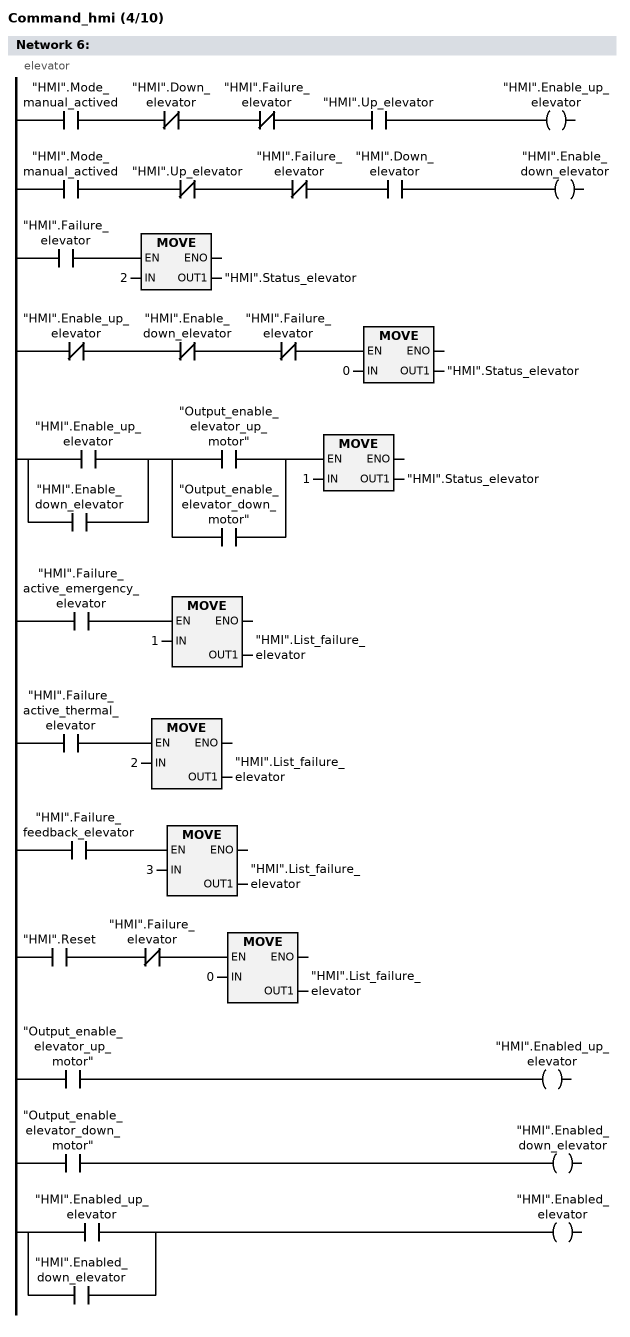
   RUNG wire#powerrail
      Contact( "HMI".Mode_manual_actived )
      I_Contact( "HMI".Down_elevator )
      I_Contact( "HMI".Failure_elevator )
      Contact( "HMI".Up_elevator )
      Coil( "HMI".Enable_up_elevator )
   END_RUNG
   RUNG wire#powerrail
      Contact( "HMI".Mode_manual_actived )
      I_Contact( "HMI".Up_elevator )
      I_Contact( "HMI".Failure_elevator )
      Contact( "HMI".Down_elevator )
      Coil( "HMI".Enable_down_elevator )
   END_RUNG
   RUNG wire#powerrail
      Contact( "HMI".Failure_elevator )
      Move(in := 2, out1 => "HMI".Status_elevator)
   END_RUNG
   RUNG wire#powerrail
      I_Contact( "HMI".Enable_up_elevator )
      I_Contact( "HMI".Enable_down_elevator )
      I_Contact( "HMI".Failure_elevator )
      Move(in := 0, out1 => "HMI".Status_elevator)
   END_RUNG
   RUNG wire#powerrail
      Contact( "HMI".Enable_up_elevator )
      wire#w1
      Contact( "Output_enable_elevator_up_motor" )
      wire#w2
      Move(in := 1, out1 => "HMI".Status_elevator)
   END_RUNG
   RUNG wire#powerrail
      Contact( "HMI".Enable_down_elevator )
   END_RUNG wire#w1
   RUNG wire#w1
      Contact( "Output_enable_elevator_down_motor" )
   END_RUNG wire#w2
   RUNG wire#powerrail
      Contact( "HMI".Failure_active_emergency_elevator )
      Move(in := 1, out1 => "HMI".List_failure_elevator)
   END_RUNG
   RUNG wire#powerrail
      Contact( "HMI".Failure_active_thermal_elevator )
      Move(in := 2, out1 => "HMI".List_failure_elevator)
   END_RUNG
   RUNG wire#powerrail
      Contact( "HMI".Failure_feedback_elevator )
      Move(in := 3, out1 => "HMI".List_failure_elevator)
   END_RUNG
   RUNG wire#powerrail
      Contact( "HMI".Reset )
      I_Contact( "HMI".Failure_elevator )
      Move(in := 0, out1 => "HMI".List_failure_elevator)
   END_RUNG
   RUNG wire#powerrail
      Contact( "Output_enable_elevator_up_motor" )
      Coil( "HMI".Enabled_up_elevator )
   END_RUNG
   RUNG wire#powerrail
      Contact( "Output_enable_elevator_down_motor" )
      Coil( "HMI".Enabled_down_elevator )
   END_RUNG
   RUNG wire#powerrail
      Contact( "HMI".Enabled_up_elevator )
      wire#w3
      Coil( "HMI".Enabled_elevator )
   END_RUNG
   RUNG wire#powerrail
      Contact( "HMI".Enabled_down_elevator )
   END_RUNG wire#w3
   // the same network as SCL:
   "HMI".Enable_up_elevator := "HMI".Mode_manual_actived AND NOT "HMI".Down_elevator AND NOT "HMI".Failure_elevator AND "HMI".Up_elevator;
   "HMI".Enable_down_elevator := "HMI".Mode_manual_actived AND NOT "HMI".Up_elevator AND NOT "HMI".Failure_elevator AND "HMI".Down_elevator;
   IF "HMI".Failure_elevator THEN "HMI".Status_elevator := 2; END_IF;
   IF NOT "HMI".Enable_up_elevator AND NOT "HMI".Enable_down_elevator AND NOT "HMI".Failure_elevator THEN
       "HMI".Status_elevator := 0;
   END_IF;
   IF ("HMI".Enable_up_elevator OR "HMI".Enable_down_elevator) AND ("Output_enable_elevator_up_motor" OR "Output_enable_elevator_down_motor") THEN
       "HMI".Status_elevator := 1;
   END_IF;
   IF "HMI".Failure_active_emergency_elevator THEN "HMI".List_failure_elevator := 1; END_IF;
   IF "HMI".Failure_active_thermal_elevator THEN "HMI".List_failure_elevator := 2; END_IF;
   IF "HMI".Failure_feedback_elevator THEN "HMI".List_failure_elevator := 3; END_IF;
   IF "HMI".Reset AND NOT "HMI".Failure_elevator THEN "HMI".List_failure_elevator := 0; END_IF;
   "HMI".Enabled_up_elevator := "Output_enable_elevator_up_motor";
   "HMI".Enabled_down_elevator := "Output_enable_elevator_down_motor";
   "HMI".Enabled_elevator := "HMI".Enabled_up_elevator OR "HMI".Enabled_down_elevator;
END_REGION

REGION Network 7
   // load pallet
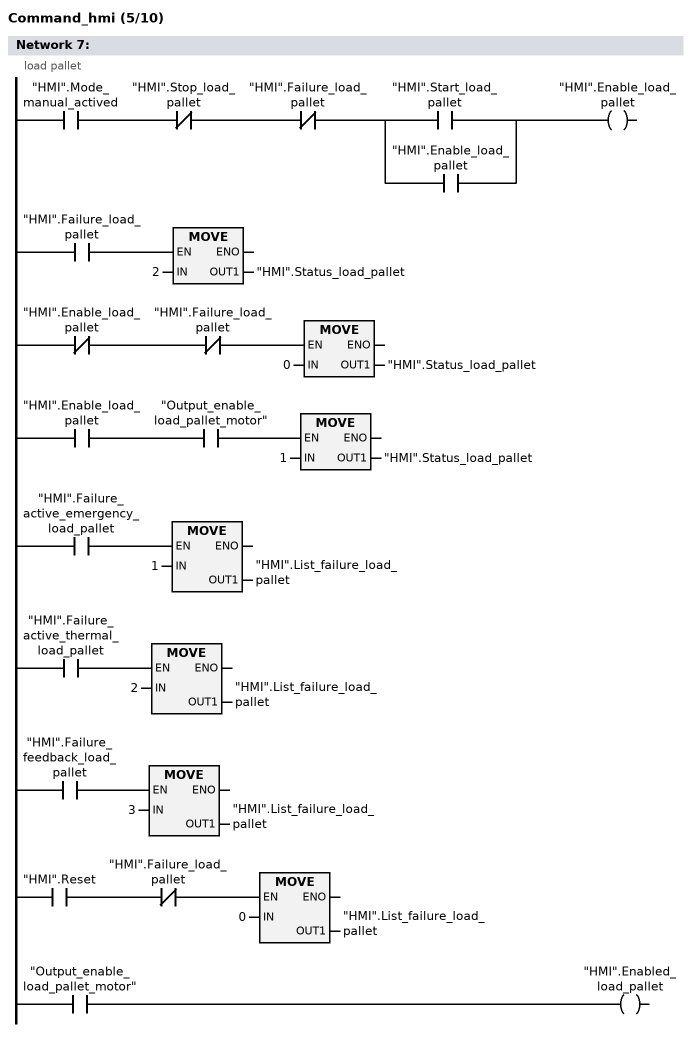
   RUNG wire#powerrail
      Contact( "HMI".Mode_manual_actived )
      I_Contact( "HMI".Stop_load_pallet )
      I_Contact( "HMI".Failure_load_pallet )
      wire#w1
      Contact( "HMI".Start_load_pallet )
      wire#w2
      Coil( "HMI".Enable_load_pallet )
   END_RUNG
   RUNG wire#w1
      Contact( "HMI".Enable_load_pallet )
   END_RUNG wire#w2
   RUNG wire#powerrail
      Contact( "HMI".Failure_load_pallet )
      Move(in := 2, out1 => "HMI".Status_load_pallet)
   END_RUNG
   RUNG wire#powerrail
      I_Contact( "HMI".Enable_load_pallet )
      I_Contact( "HMI".Failure_load_pallet )
      Move(in := 0, out1 => "HMI".Status_load_pallet)
   END_RUNG
   RUNG wire#powerrail
      Contact( "HMI".Enable_load_pallet )
      Contact( "Output_enable_load_pallet_motor" )
      Move(in := 1, out1 => "HMI".Status_load_pallet)
   END_RUNG
   RUNG wire#powerrail
      Contact( "HMI".Failure_active_emergency_load_pallet )
      Move(in := 1, out1 => "HMI".List_failure_load_pallet)
   END_RUNG
   RUNG wire#powerrail
      Contact( "HMI".Failure_active_thermal_load_pallet )
      Move(in := 2, out1 => "HMI".List_failure_load_pallet)
   END_RUNG
   RUNG wire#powerrail
      Contact( "HMI".Failure_feedback_load_pallet )
      Move(in := 3, out1 => "HMI".List_failure_load_pallet)
   END_RUNG
   RUNG wire#powerrail
      Contact( "HMI".Reset )
      I_Contact( "HMI".Failure_load_pallet )
      Move(in := 0, out1 => "HMI".List_failure_load_pallet)
   END_RUNG
   RUNG wire#powerrail
      Contact( "Output_enable_load_pallet_motor" )
      Coil( "HMI".Enabled_load_pallet )
   END_RUNG
   // the same network as SCL:
   "HMI".Enable_load_pallet := "HMI".Mode_manual_actived AND NOT "HMI".Stop_load_pallet AND NOT "HMI".Failure_load_pallet AND ("HMI".Start_load_pallet OR "HMI".Enable_load_pallet);
   IF "HMI".Failure_load_pallet THEN "HMI".Status_load_pallet := 2; END_IF;
   IF NOT "HMI".Enable_load_pallet AND NOT "HMI".Failure_load_pallet THEN
       "HMI".Status_load_pallet := 0;
   END_IF;
   IF "HMI".Enable_load_pallet AND "Output_enable_load_pallet_motor" THEN
       "HMI".Status_load_pallet := 1;
   END_IF;
   IF "HMI".Failure_active_emergency_load_pallet THEN "HMI".List_failure_load_pallet := 1; END_IF;
   IF "HMI".Failure_active_thermal_load_pallet THEN "HMI".List_failure_load_pallet := 2; END_IF;
   IF "HMI".Failure_feedback_load_pallet THEN "HMI".List_failure_load_pallet := 3; END_IF;
   IF "HMI".Reset AND NOT "HMI".Failure_load_pallet THEN "HMI".List_failure_load_pallet := 0; END_IF;
   "HMI".Enabled_load_pallet := "Output_enable_load_pallet_motor";
END_REGION

REGION Network 8
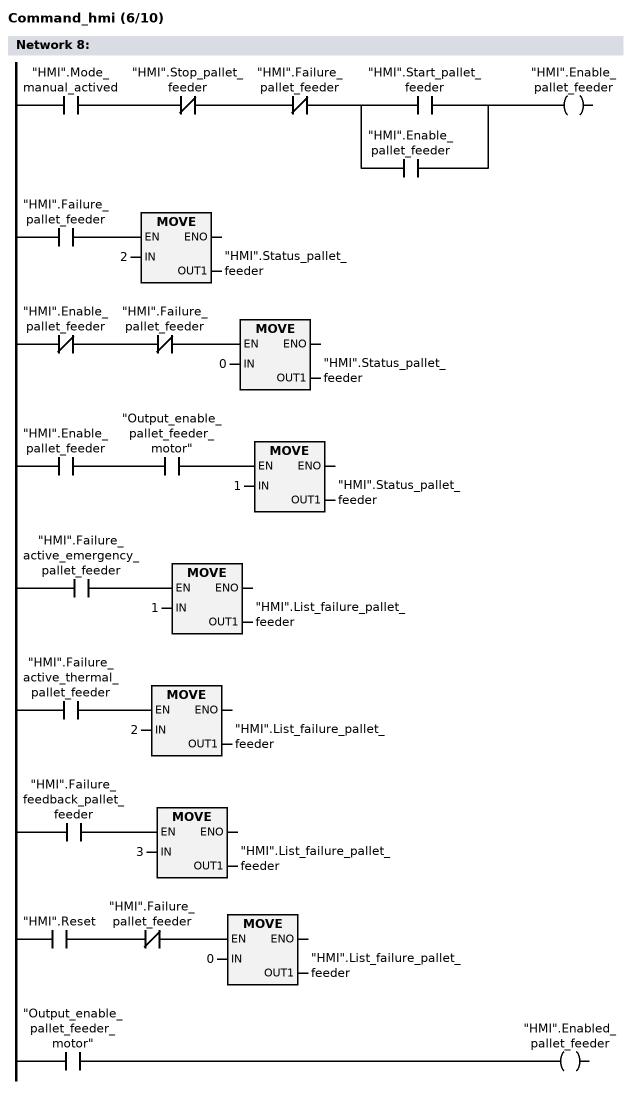
   RUNG wire#powerrail
      Contact( "HMI".Mode_manual_actived )
      I_Contact( "HMI".Stop_pallet_feeder )
      I_Contact( "HMI".Failure_pallet_feeder )
      wire#w1
      Contact( "HMI".Start_pallet_feeder )
      wire#w2
      Coil( "HMI".Enable_pallet_feeder )
   END_RUNG
   RUNG wire#w1
      Contact( "HMI".Enable_pallet_feeder )
   END_RUNG wire#w2
   RUNG wire#powerrail
      Contact( "HMI".Failure_pallet_feeder )
      Move(in := 2, out1 => "HMI".Status_pallet_feeder)
   END_RUNG
   RUNG wire#powerrail
      I_Contact( "HMI".Enable_pallet_feeder )
      I_Contact( "HMI".Failure_pallet_feeder )
      Move(in := 0, out1 => "HMI".Status_pallet_feeder)
   END_RUNG
   RUNG wire#powerrail
      Contact( "HMI".Enable_pallet_feeder )
      Contact( "Output_enable_pallet_feeder_motor" )
      Move(in := 1, out1 => "HMI".Status_pallet_feeder)
   END_RUNG
   RUNG wire#powerrail
      Contact( "HMI".Failure_active_emergency_pallet_feeder )
      Move(in := 1, out1 => "HMI".List_failure_pallet_feeder)
   END_RUNG
   RUNG wire#powerrail
      Contact( "HMI".Failure_active_thermal_pallet_feeder )
      Move(in := 2, out1 => "HMI".List_failure_pallet_feeder)
   END_RUNG
   RUNG wire#powerrail
      Contact( "HMI".Failure_feedback_pallet_feeder )
      Move(in := 3, out1 => "HMI".List_failure_pallet_feeder)
   END_RUNG
   RUNG wire#powerrail
      Contact( "HMI".Reset )
      I_Contact( "HMI".Failure_pallet_feeder )
      Move(in := 0, out1 => "HMI".List_failure_pallet_feeder)
   END_RUNG
   RUNG wire#powerrail
      Contact( "Output_enable_pallet_feeder_motor" )
      Coil( "HMI".Enabled_pallet_feeder )
   END_RUNG
   // the same network as SCL:
   "HMI".Enable_pallet_feeder := "HMI".Mode_manual_actived AND NOT "HMI".Stop_pallet_feeder AND NOT "HMI".Failure_pallet_feeder AND ("HMI".Start_pallet_feeder OR "HMI".Enable_pallet_feeder);
   IF "HMI".Failure_pallet_feeder THEN "HMI".Status_pallet_feeder := 2; END_IF;
   IF NOT "HMI".Enable_pallet_feeder AND NOT "HMI".Failure_pallet_feeder THEN
       "HMI".Status_pallet_feeder := 0;
   END_IF;
   IF "HMI".Enable_pallet_feeder AND "Output_enable_pallet_feeder_motor" THEN
       "HMI".Status_pallet_feeder := 1;
   END_IF;
   IF "HMI".Failure_active_emergency_pallet_feeder THEN "HMI".List_failure_pallet_feeder := 1; END_IF;
   IF "HMI".Failure_active_thermal_pallet_feeder THEN "HMI".List_failure_pallet_feeder := 2; END_IF;
   IF "HMI".Failure_feedback_pallet_feeder THEN "HMI".List_failure_pallet_feeder := 3; END_IF;
   IF "HMI".Reset AND NOT "HMI".Failure_pallet_feeder THEN "HMI".List_failure_pallet_feeder := 0; END_IF;
   "HMI".Enabled_pallet_feeder := "Output_enable_pallet_feeder_motor";
END_REGION

REGION Network 9
   // exit conveyor
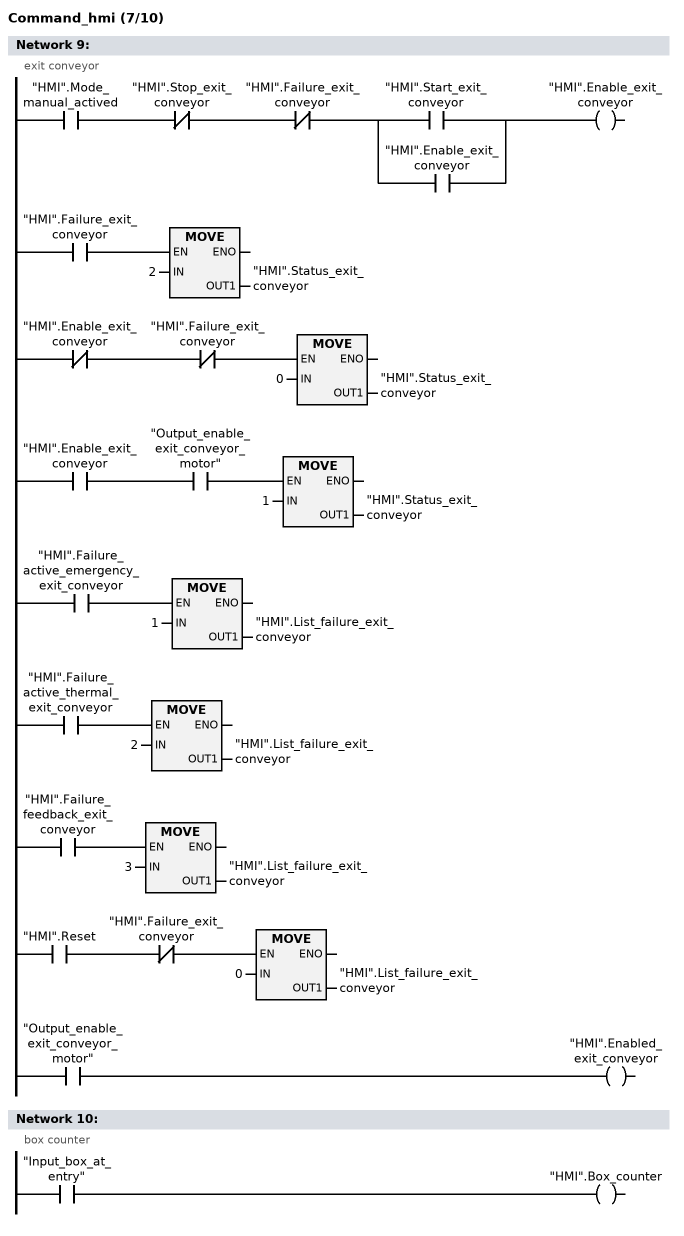
   RUNG wire#powerrail
      Contact( "HMI".Mode_manual_actived )
      I_Contact( "HMI".Stop_exit_conveyor )
      I_Contact( "HMI".Failure_exit_conveyor )
      wire#w1
      Contact( "HMI".Start_exit_conveyor )
      wire#w2
      Coil( "HMI".Enable_exit_conveyor )
   END_RUNG
   RUNG wire#w1
      Contact( "HMI".Enable_exit_conveyor )
   END_RUNG wire#w2
   RUNG wire#powerrail
      Contact( "HMI".Failure_exit_conveyor )
      Move(in := 2, out1 => "HMI".Status_exit_conveyor)
   END_RUNG
   RUNG wire#powerrail
      I_Contact( "HMI".Enable_exit_conveyor )
      I_Contact( "HMI".Failure_exit_conveyor )
      Move(in := 0, out1 => "HMI".Status_exit_conveyor)
   END_RUNG
   RUNG wire#powerrail
      Contact( "HMI".Enable_exit_conveyor )
      Contact( "Output_enable_exit_conveyor_motor" )
      Move(in := 1, out1 => "HMI".Status_exit_conveyor)
   END_RUNG
   RUNG wire#powerrail
      Contact( "HMI".Failure_active_emergency_exit_conveyor )
      Move(in := 1, out1 => "HMI".List_failure_exit_conveyor)
   END_RUNG
   RUNG wire#powerrail
      Contact( "HMI".Failure_active_thermal_exit_conveyor )
      Move(in := 2, out1 => "HMI".List_failure_exit_conveyor)
   END_RUNG
   RUNG wire#powerrail
      Contact( "HMI".Failure_feedback_exit_conveyor )
      Move(in := 3, out1 => "HMI".List_failure_exit_conveyor)
   END_RUNG
   RUNG wire#powerrail
      Contact( "HMI".Reset )
      I_Contact( "HMI".Failure_exit_conveyor )
      Move(in := 0, out1 => "HMI".List_failure_exit_conveyor)
   END_RUNG
   RUNG wire#powerrail
      Contact( "Output_enable_exit_conveyor_motor" )
      Coil( "HMI".Enabled_exit_conveyor )
   END_RUNG
   // the same network as SCL:
   "HMI".Enable_exit_conveyor := "HMI".Mode_manual_actived AND NOT "HMI".Stop_exit_conveyor AND NOT "HMI".Failure_exit_conveyor AND ("HMI".Start_exit_conveyor OR "HMI".Enable_exit_conveyor);
   IF "HMI".Failure_exit_conveyor THEN "HMI".Status_exit_conveyor := 2; END_IF;
   IF NOT "HMI".Enable_exit_conveyor AND NOT "HMI".Failure_exit_conveyor THEN
       "HMI".Status_exit_conveyor := 0;
   END_IF;
   IF "HMI".Enable_exit_conveyor AND "Output_enable_exit_conveyor_motor" THEN
       "HMI".Status_exit_conveyor := 1;
   END_IF;
   IF "HMI".Failure_active_emergency_exit_conveyor THEN "HMI".List_failure_exit_conveyor := 1; END_IF;
   IF "HMI".Failure_active_thermal_exit_conveyor THEN "HMI".List_failure_exit_conveyor := 2; END_IF;
   IF "HMI".Failure_feedback_exit_conveyor THEN "HMI".List_failure_exit_conveyor := 3; END_IF;
   IF "HMI".Reset AND NOT "HMI".Failure_exit_conveyor THEN "HMI".List_failure_exit_conveyor := 0; END_IF;
   "HMI".Enabled_exit_conveyor := "Output_enable_exit_conveyor_motor";
END_REGION

REGION Network 10
   // box counter
   RUNG wire#powerrail
      Contact( "Input_box_at_entry" )
      Coil( "HMI".Box_counter )
   END_RUNG
   // the same network as SCL:
   "HMI".Box_counter := "Input_box_at_entry";
END_REGION

REGION Network 11
   // Enabled turn
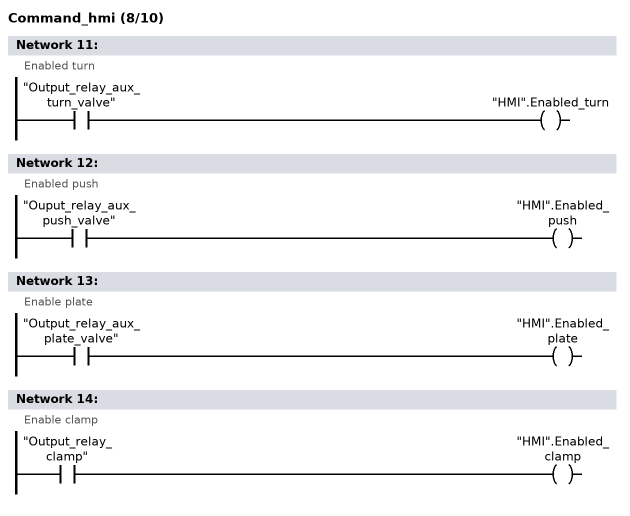
   RUNG wire#powerrail
      Contact( "Output_relay_aux_turn_valve" )
      Coil( "HMI".Enabled_turn )
   END_RUNG
   // the same network as SCL:
   "HMI".Enabled_turn := "Output_relay_aux_turn_valve";
END_REGION

REGION Network 12
   // Enabled push
   RUNG wire#powerrail
      Contact( "Ouput_relay_aux_push_valve" )
      Coil( "HMI".Enabled_push )
   END_RUNG
   // the same network as SCL:
   "HMI".Enabled_push := "Ouput_relay_aux_push_valve";
END_REGION

REGION Network 13
   // Enable plate
   RUNG wire#powerrail
      Contact( "Output_relay_aux_plate_valve" )
      Coil( "HMI".Enabled_plate )
   END_RUNG
   // the same network as SCL:
   "HMI".Enabled_plate := "Output_relay_aux_plate_valve";
END_REGION

REGION Network 14
   // Enable clamp
   RUNG wire#powerrail
      Contact( "Output_relay_clamp" )
      Coil( "HMI".Enabled_clamp )
   END_RUNG
   // the same network as SCL:
   "HMI".Enabled_clamp := "Output_relay_clamp";
END_REGION

REGION Network 15
   // elevator moving
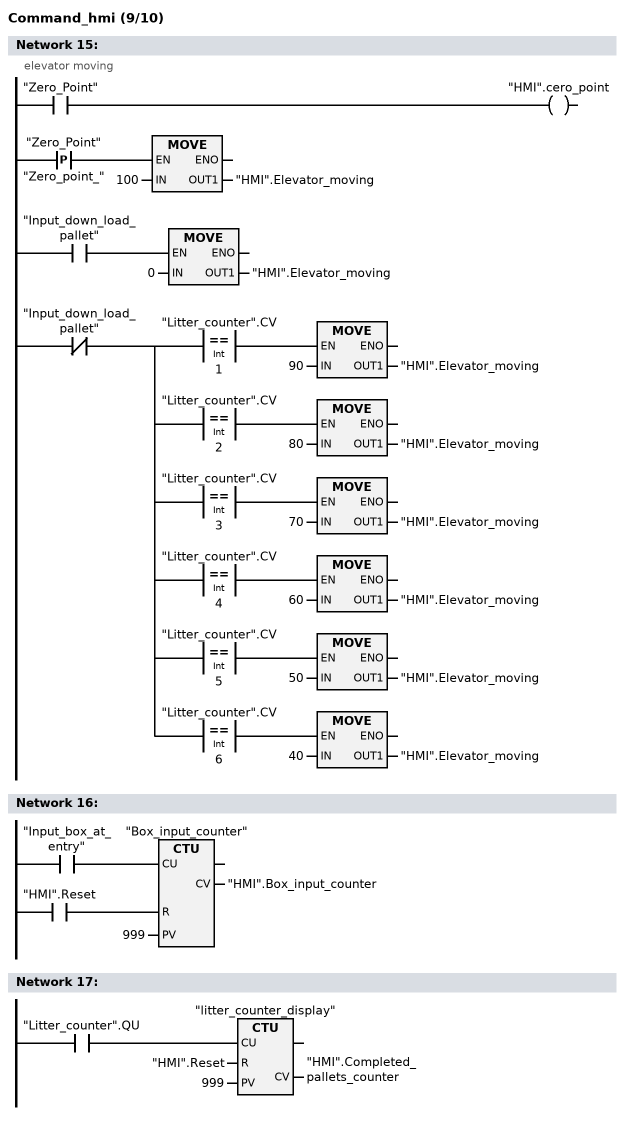
   RUNG wire#powerrail
      Contact( "Zero_Point" )
      Coil( "HMI".cero_point )
   END_RUNG
   RUNG wire#powerrail
      P_Contact(operand := "Zero_Point", bit := "Zero_point_")
      Move(in := 100, out1 => "HMI".Elevator_moving)
   END_RUNG
   RUNG wire#powerrail
      Contact( "Input_down_load_pallet" )
      Move(in := 0, out1 => "HMI".Elevator_moving)
   END_RUNG
   RUNG wire#powerrail
      I_Contact( "Input_down_load_pallet" )
      wire#w1
      { S7_Templates := "SrcType := Int" } EQ_Contact(in1 := "Litter_counter".CV, in2 := 1)
      Move(in := 90, out1 => "HMI".Elevator_moving)
   END_RUNG
   RUNG wire#w1
      { S7_Templates := "SrcType := Int" } EQ_Contact(in1 := "Litter_counter".CV, in2 := 2)
      Move(in := 80, out1 => "HMI".Elevator_moving)
   END_RUNG
   RUNG wire#w1
      { S7_Templates := "SrcType := Int" } EQ_Contact(in1 := "Litter_counter".CV, in2 := 3)
      Move(in := 70, out1 => "HMI".Elevator_moving)
   END_RUNG
   RUNG wire#w1
      { S7_Templates := "SrcType := Int" } EQ_Contact(in1 := "Litter_counter".CV, in2 := 4)
      Move(in := 60, out1 => "HMI".Elevator_moving)
   END_RUNG
   RUNG wire#w1
      { S7_Templates := "SrcType := Int" } EQ_Contact(in1 := "Litter_counter".CV, in2 := 5)
      Move(in := 50, out1 => "HMI".Elevator_moving)
   END_RUNG
   RUNG wire#w1
      { S7_Templates := "SrcType := Int" } EQ_Contact(in1 := "Litter_counter".CV, in2 := 6)
      Move(in := 40, out1 => "HMI".Elevator_moving)
   END_RUNG
   // the same network as SCL:
   "HMI".cero_point := "Zero_Point";
   #_w1 := "Zero_Point" AND NOT "Zero_point_";   // rising edge of "Zero_Point"
   "Zero_point_" := "Zero_Point";
   IF #_w1 THEN "HMI".Elevator_moving := 100; END_IF;
   IF "Input_down_load_pallet" THEN "HMI".Elevator_moving := 0; END_IF;
   #_w2 := NOT "Input_down_load_pallet";
   IF #_w2 AND ("Litter_counter".CV = 1) THEN "HMI".Elevator_moving := 90; END_IF;
   IF #_w2 AND ("Litter_counter".CV = 2) THEN "HMI".Elevator_moving := 80; END_IF;
   IF #_w2 AND ("Litter_counter".CV = 3) THEN "HMI".Elevator_moving := 70; END_IF;
   IF #_w2 AND ("Litter_counter".CV = 4) THEN "HMI".Elevator_moving := 60; END_IF;
   IF #_w2 AND ("Litter_counter".CV = 5) THEN "HMI".Elevator_moving := 50; END_IF;
   IF #_w2 AND ("Litter_counter".CV = 6) THEN "HMI".Elevator_moving := 40; END_IF;
END_REGION

REGION Network 16
   "Box_input_counter".CTU(CU := "Input_box_at_entry",
                           R := "HMI".Reset,
                           PV := 999,
                           CV => "HMI".Box_input_counter);
END_REGION

REGION Network 17
   "litter_counter_display".CTU(CU := "Litter_counter".QU,
                           R := "HMI".Reset,
                           PV := 999,
                           CV => "HMI".Completed_pallets_counter);
END_REGION

REGION Network 18
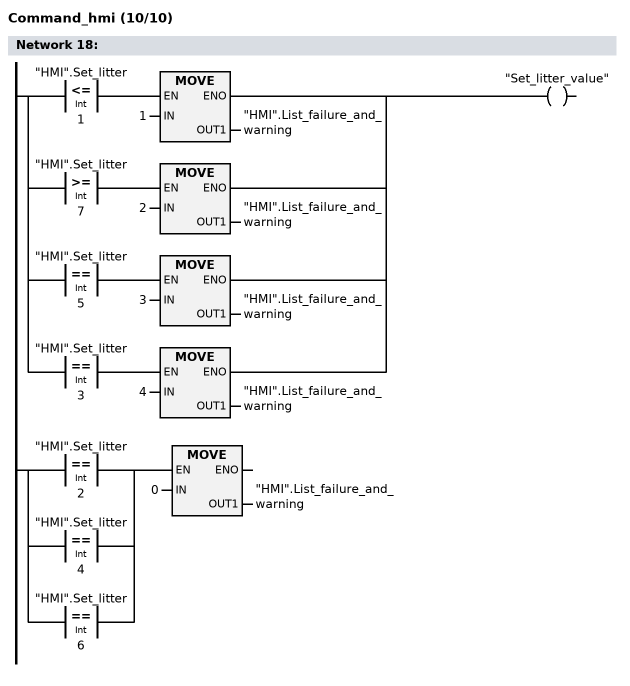
   RUNG wire#powerrail
      { S7_Templates := "SrcType := Int" } LE_Contact(in1 := "HMI".Set_litter, in2 := 1)
      Move(in := 1, out1 => "HMI".List_failure_and_warning)
      wire#w1
      Coil( "Set_litter_value" )
   END_RUNG
   RUNG wire#powerrail
      { S7_Templates := "SrcType := Int" } GE_Contact(in1 := "HMI".Set_litter, in2 := 7)
      Move(in := 2, out1 => "HMI".List_failure_and_warning)
   END_RUNG wire#w1
   RUNG wire#powerrail
      { S7_Templates := "SrcType := Int" } EQ_Contact(in1 := "HMI".Set_litter, in2 := 5)
      Move(in := 3, out1 => "HMI".List_failure_and_warning)
   END_RUNG wire#w1
   RUNG wire#powerrail
      { S7_Templates := "SrcType := Int" } EQ_Contact(in1 := "HMI".Set_litter, in2 := 3)
      Move(in := 4, out1 => "HMI".List_failure_and_warning)
   END_RUNG wire#w1
   RUNG wire#powerrail
      { S7_Templates := "SrcType := Int" } EQ_Contact(in1 := "HMI".Set_litter, in2 := 2)
      wire#w2
      Move(in := 0, out1 => "HMI".List_failure_and_warning)
   END_RUNG
   RUNG wire#powerrail
      { S7_Templates := "SrcType := Int" } EQ_Contact(in1 := "HMI".Set_litter, in2 := 4)
   END_RUNG wire#w2
   RUNG wire#powerrail
      { S7_Templates := "SrcType := Int" } EQ_Contact(in1 := "HMI".Set_litter, in2 := 6)
   END_RUNG wire#w2
   // the same network as SCL:
   #_w1 := "HMI".Set_litter <= 1;
   IF #_w1 THEN "HMI".List_failure_and_warning := 1; END_IF;
   #_w2 := "HMI".Set_litter >= 7;
   IF #_w2 THEN "HMI".List_failure_and_warning := 2; END_IF;
   #_w3 := "HMI".Set_litter = 5;
   IF #_w3 THEN "HMI".List_failure_and_warning := 3; END_IF;
   #_w4 := "HMI".Set_litter = 3;
   IF #_w4 THEN "HMI".List_failure_and_warning := 4; END_IF;
   "Set_litter_value" := #_w1 OR #_w2 OR #_w3 OR #_w4;
   IF ("HMI".Set_litter = 2) OR ("HMI".Set_litter = 4) OR ("HMI".Set_litter = 6) THEN
       "HMI".List_failure_and_warning := 0;
   END_IF;
END_REGION
END_FUNCTION

FUNCTION "MHJ-PLC-Lab-Function-S71200" : Void   // FC9000, SCL
{ S7_Optimized_Access := 'TRUE' }
VERSION : 0.1
   VAR_TEMP
      rdTimeReturn : Int;
      outputTime : DTL;
      SyncVal : Byte;
      forVal : Int;
      forVal_2 : Int;
      Value : Byte;
   END_VAR
   VAR CONSTANT
      CompVal : Byte := 16#34;
      Value_01 : Byte := 16#11;
      Value_01_DW : DWord := 16#A165_D992;
      Value_02_DW : DWord := 16#58BE_4401;
   END_VAR
BEGIN

   #Value:=PEEK(area := 16#82,
        dbNumber := 0,
        byteOffset := 511);
   #Value := #Value + 1;

   POKE(area := 16#82,
        dbNumber := 0,
        byteOffset := 511,
        value := #Value);

   POKE(area:=16#81,
        dbNumber:=0,
        byteOffset:=1016,
        value:=#Value_01_DW);
   POKE(area := 16#81,
        dbNumber := 0,
        byteOffset := 1020,
        value := #Value_02_DW);

   POKE(area := 16#81,
        dbNumber := 0,
        byteOffset := 511,
        value := B#16#00);

   FOR #forVal := 0 TO 120 DO
       FOR #forVal_2:=0 TO 10 DO
           #rdTimeReturn:=RD_SYS_T(#outputTime);
           #rdTimeReturn := WR_SYS_T(#outputTime);
           #rdTimeReturn := RD_SYS_T(#outputTime);
           #rdTimeReturn := WR_SYS_T(#outputTime);
       END_FOR;
       #SyncVal:= PEEK(area := 16#81,
                      dbNumber := 0,
                      byteOffset := 511);
       IF #SyncVal = #CompVal THEN
          GOTO M_1;
       END_IF;
   END_FOR;
   RETURN;

   M_1:
   POKE(area := 16#81,
        dbNumber := 0,
        byteOffset := 511,
        value := B#16#0);
END_FUNCTION

ORGANIZATION_BLOCK "Main"   // OB1, LAD, ProgramCycle
TITLE = "Main Program Sweep (Cycle)"
{ S7_Optimized_Access := 'TRUE' }
VERSION : 0.1
   VAR_INPUT
      Initial_Call : Bool;   // Initial call of this OB
      Remanence : Bool;   // =True, if remanent data are available
   END_VAR
BEGIN

REGION Network 1: FACTORY IO MODULE
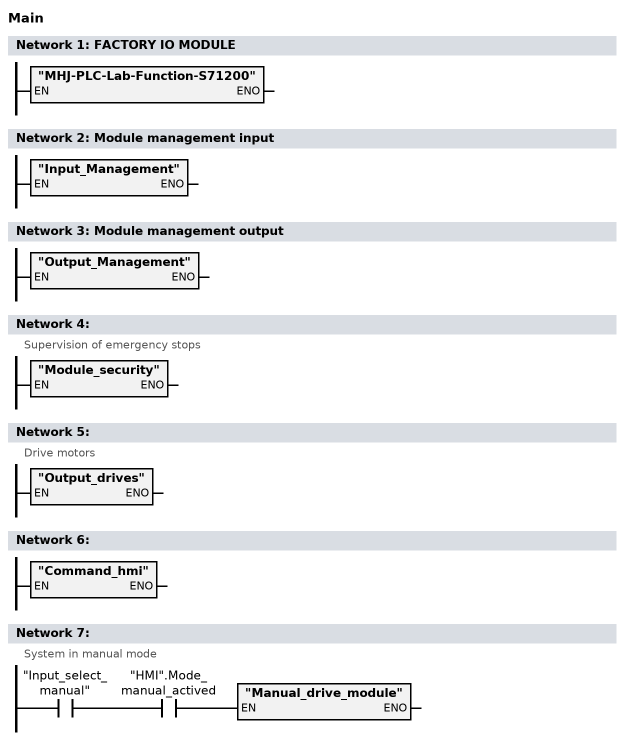
   RUNG wire#powerrail
      "MHJ-PLC-Lab-Function-S71200"()
   END_RUNG
   // the same network as SCL:
   "MHJ-PLC-Lab-Function-S71200"();
END_REGION

REGION Network 2: Module management input
   RUNG wire#powerrail
      "Input_Management"()
   END_RUNG
   // the same network as SCL:
   "Input_Management"();
END_REGION

REGION Network 3: Module management output
   RUNG wire#powerrail
      "Output_Management"()
   END_RUNG
   // the same network as SCL:
   "Output_Management"();
END_REGION

REGION Network 4
   // Supervision of emergency stops
   RUNG wire#powerrail
      "Module_security"()
   END_RUNG
   // the same network as SCL:
   "Module_security"();
END_REGION

REGION Network 5
   // Drive motors
   RUNG wire#powerrail
      "Output_drives"()
   END_RUNG
   // the same network as SCL:
   "Output_drives"();
END_REGION

REGION Network 6
   RUNG wire#powerrail
      "Command_hmi"()
   END_RUNG
   // the same network as SCL:
   "Command_hmi"();
END_REGION

REGION Network 7
   // System in manual mode
   RUNG wire#powerrail
      Contact( "Input_select_manual" )
      Contact( "HMI".Mode_manual_actived )
      "Manual_drive_module"()
   END_RUNG
   // the same network as SCL:
   IF "Input_select_manual" AND "HMI".Mode_manual_actived THEN "Manual_drive_module"(); END_IF;
END_REGION
END_ORGANIZATION_BLOCK

(* ===== HMI "HMI_RT_1" =====
system functions are stored by id; their names below are inferred from use
connection "HMI_Connection_1": ETHERNET, SMART_S7_1200_OMS

HMI tags "Default tag table"
   "Mode_manual" : Bool = PLC HMI.Mode_manual AT %DB28.DBX0.0, 1 s
   "Mode_Auto" : Bool = PLC HMI.Mode_auto AT %DB28.DBX0.1, 1 s
   "List_message" : Int = PLC HMI.List_status AT %DB28.DBW2, 1 s
   "Mode_manual_actived" : Bool = PLC HMI.Mode_manual_actived AT %DB28.DBX0.2, 1 s
   "Mode_auto_actived" : Bool = PLC HMI.Mode_auto_actived AT %DB28.DBX0.3, 1 s
   "Mode_rest" : Bool = PLC HMI.Mode_rest AT %DB28.DBX0.4, 1 s
   "Start_box_feeder" : Bool = PLC HMI.Start_box_feeder AT %DB28.DBX4.0, 1 s
   "Stop_box_feeder" : Bool = PLC HMI.Stop_box_feeder AT %DB28.DBX4.1, 1 s
   "Failure_active_emergency_box_feeder" : Bool = PLC HMI.Failure_active_emergency_box_feeder AT %DB28.DBX4.4, 1 s
   "Failure_active_thermal_box_feeder" : Bool = PLC HMI.Failure_active_thermal_box_feeder AT %DB28.DBX4.5, 1 s
   "Failure_feedback_box_feeder" : Bool = PLC HMI.Failure_feedback_box_feeder AT %DB28.DBX4.6, 1 s
   "Enable_box_feeder" : Bool = PLC HMI.Enable_box_feeder AT %DB28.DBX4.2, 1 s
   "Failure_box_feeder" : Bool = PLC HMI.Failure_box_feeder AT %DB28.DBX4.7, 1 s
   "Status_box_feeder" : Int = PLC HMI.Status_box_feeder AT %DB28.DBW6, 1 s
   "Reset" : Bool = PLC HMI.Reset AT %DB28.DBX0.5, 1 s
   "List_failure_box_feeder" : Int = PLC HMI.List_failure_box_feeder AT %DB28.DBW8, 1 s
   "Rotation_box_feeder" : Int = PLC HMI.Rotation_box_feeder AT %DB28.DBW10, 1 s
   "Start_load_beld" : Bool = PLC HMI.Start_load_beld AT %DB28.DBX12.0, 1 s
   "Stop_load_beld" : Bool = PLC HMI.Stop_load_beld AT %DB28.DBX12.1, 1 s
   "Enable_load_beld" : Bool = PLC HMI.Enable_load_beld AT %DB28.DBX12.2, 1 s
   "Failure_active_emergency_load_beld" : Bool = PLC HMI.Failure_active_emergency_load_beld AT %DB28.DBX12.4, 1 s
   "Failure_active_thermal_load_beld" : Bool = PLC HMI.Failure_active_thermal_load_beld AT %DB28.DBX12.5, 1 s
   "Failure_feedback_load_beld" : Bool = PLC HMI.Failure_feedback_load_beld AT %DB28.DBX12.6, 1 s
   "Failure_load_beld" : Bool = PLC HMI.Failure_load_beld AT %DB28.DBX12.7, 1 s
   "Status_load_beld" : Int = PLC HMI.Status_load_beld AT %DB28.DBW14, 1 s
   "List_failure_load_beld" : Int = PLC HMI.List_failure_load_beld AT %DB28.DBW16, 1 s
   "Rotation_load_beld" : Int = PLC HMI.Rotation_load_beld AT %DB28.DBW18, 1 s
   "Up_elevator" : Bool = PLC HMI.Up_elevator AT %DB28.DBX20.0, 1 s
   "Down_elevator" : Bool = PLC HMI.Down_elevator AT %DB28.DBX20.1, 1 s
   "Enable_up_elevator" : Bool = PLC HMI.Enable_up_elevator AT %DB28.DBX20.2, 1 s
   "Enable_down_elevator" : Bool = PLC HMI.Enable_down_elevator AT %DB28.DBX20.3, 1 s
   "Failure_active_emergency_elevator" : Bool = PLC HMI.Failure_active_emergency_elevator AT %DB28.DBX20.7, 1 s
   "Failure_active_thermal_elevator" : Bool = PLC HMI.Failure_active_thermal_elevator AT %DB28.DBX21.0, 1 s
   "Failure_feedback_elevator" : Bool = PLC HMI.Failure_feedback_elevator AT %DB28.DBX21.1, 1 s
   "Failure_elevator" : Bool = PLC HMI.Failure_elevator AT %DB28.DBX21.2, 1 s
   "Status_elevator" : Int = PLC HMI.Status_elevator AT %DB28.DBW22, 1 s
   "List_failure_elevator" : Int = PLC HMI.List_failure_elevator AT %DB28.DBW24, 1 s
   "Rotation_elevator" : Int = PLC HMI.Rotation_elevator AT %DB28.DBW26, 1 s
   "Start_load_pallet" : Bool = PLC HMI.Start_load_pallet AT %DB28.DBX28.0, 1 s
   "Stop_load_pallet" : Bool = PLC HMI.Stop_load_pallet AT %DB28.DBX28.1, 1 s
   "Enable_load_pallet" : Bool = PLC HMI.Enable_load_pallet AT %DB28.DBX28.2, 1 s
   "Failure_active_emergency_load_pallet" : Bool = PLC HMI.Failure_active_emergency_load_pallet AT %DB28.DBX28.4, 1 s
   "Failure_active_thermal_load_pallet" : Bool = PLC HMI.Failure_active_thermal_load_pallet AT %DB28.DBX28.5, 1 s
   "Failure_feedback_load_pallet" : Bool = PLC HMI.Failure_feedback_load_pallet AT %DB28.DBX28.6, 1 s
   "Failure_load_pallet" : Bool = PLC HMI.Failure_load_pallet AT %DB28.DBX28.7, 1 s
   "Status_load_pallet" : Int = PLC HMI.Status_load_pallet AT %DB28.DBW30, 1 s
   "List_failure_load_pallet" : Int = PLC HMI.List_failure_load_pallet AT %DB28.DBW32, 1 s
   "Rotation_load_pallet" : Int = PLC HMI.Rotation_load_pallet AT %DB28.DBW34, 1 s
   "Start_pallet_feeder" : Bool = PLC HMI.Start_pallet_feeder AT %DB28.DBX36.0, 1 s
   "Stop_pallet_feeder" : Bool = PLC HMI.Stop_pallet_feeder AT %DB28.DBX36.1, 1 s
   "Enable_pallet_feeder" : Bool = PLC HMI.Enable_pallet_feeder AT %DB28.DBX36.2, 1 s
   "Failure_active_emergency_pallet_feeder" : Bool = PLC HMI.Failure_active_emergency_pallet_feeder AT %DB28.DBX36.4, 1 s
   "Failure_active_thermal_pallet_feeder" : Bool = PLC HMI.Failure_active_thermal_pallet_feeder AT %DB28.DBX36.5, 1 s
   "Failure_feedback_pallet_feeder" : Bool = PLC HMI.Failure_feedback_pallet_feeder AT %DB28.DBX36.6, 1 s
   "Failure_pallet_feeder" : Bool = PLC HMI.Failure_pallet_feeder AT %DB28.DBX36.7, 1 s
   "Status_pallet_feeder" : Int = PLC HMI.Status_pallet_feeder AT %DB28.DBW38, 1 s
   "List_failure_pallet_feeder" : Int = PLC HMI.List_failure_pallet_feeder AT %DB28.DBW40, 1 s
   "Rotation_pallet_feeder" : Int = PLC HMI.Rotation_pallet_feeder AT %DB28.DBW42, 1 s
   "Start_exit_conveyor" : Bool = PLC HMI.Start_exit_conveyor AT %DB28.DBX44.0, 1 s
   "Stop_exit_conveyor" : Bool = PLC HMI.Stop_exit_conveyor AT %DB28.DBX44.1, 1 s
   "Enable_exit_conveyor" : Bool = PLC HMI.Enable_exit_conveyor AT %DB28.DBX44.2, 1 s
   "Failure_active_emergency_exit_conveyor" : Bool = PLC HMI.Failure_active_emergency_exit_conveyor AT %DB28.DBX44.4, 1 s
   "Failure_active_thermal_exit_conveyor" : Bool = PLC HMI.Failure_active_thermal_exit_conveyor AT %DB28.DBX44.5, 1 s
   "Failure_feedback_exit_conveyor" : Bool = PLC HMI.Failure_feedback_exit_conveyor AT %DB28.DBX44.6, 1 s
   "Failure_exit_conveyor" : Bool = PLC HMI.Failure_exit_conveyor AT %DB28.DBX44.7, 1 s
   "Status_exit_conveyor" : Int = PLC HMI.Status_exit_conveyor AT %DB28.DBW46, 1 s
   "List_failure_exit_conveyor" : Int = PLC HMI.List_failure_exit_conveyor AT %DB28.DBW48, 1 s
   "Rotation_exit_conveyor" : Int = PLC HMI.Rotation_exit_conveyor AT %DB28.DBW50, 1 s
   "Enable_turn" : Bool = PLC HMI.Enable_turn AT %DB28.DBX52.0, 1 s
   "Enable_push" : Bool = PLC HMI.Enable_push AT %DB28.DBX52.2, 1 s
   "Enable_plate" : Bool = PLC HMI.Enable_plate AT %DB28.DBX52.4, 1 s
   "Enable_clamp" : Bool = PLC HMI.Enable_clamp AT %DB28.DBX52.6, 1 s
   "Enabled_box_feeder" : Bool = PLC HMI.Enabled_box_feeder AT %DB28.DBX4.3, 1 s
   "Enabled_clamp" : Bool = PLC HMI.Enabled_clamp AT %DB28.DBX52.7, 1 s
   "Enabled_up_elevator" : Bool = PLC HMI.Enabled_up_elevator AT %DB28.DBX20.4, 1 s
   "Enabled_turn" : Bool = PLC HMI.Enabled_turn AT %DB28.DBX52.1, 1 s
   "Enabled_push" : Bool = PLC HMI.Enabled_push AT %DB28.DBX52.3, 1 s
   "Enabled_plate" : Bool = PLC HMI.Enabled_plate AT %DB28.DBX52.5, 1 s
   "Enabled_pallet_feeder" : Bool = PLC HMI.Enabled_pallet_feeder AT %DB28.DBX36.3, 1 s
   "Enabled_load_pallet" : Bool = PLC HMI.Enabled_load_pallet AT %DB28.DBX28.3, 1 s
   "Enabled_load_beld" : Bool = PLC HMI.Enabled_load_beld AT %DB28.DBX12.3, 1 s
   "Enabled_exit_conveyor" : Bool = PLC HMI.Enabled_exit_conveyor AT %DB28.DBX44.3, 1 s
   "Enabled_down_elevator" : Bool = PLC HMI.Enabled_down_elevator AT %DB28.DBX20.5, 1 s
   "Enabled_elevator" : Bool = PLC HMI.Enabled_elevator AT %DB28.DBX20.6, 1 s
   "Box_counter" : Bool = PLC HMI.Box_counter AT %DB28.DBX53.0, 1 s
   "cero_point" : Bool = PLC HMI.cero_point AT %DB28.DBX53.1, 1 s
   "Elevator_moving" : Int = PLC HMI.Elevator_moving AT %DB28.DBW54, 1 s
   "Set_box" : Int = PLC HMI.Set_box AT %DB28.DBW56, 1 s
   "Set_litter" : Int = PLC HMI.Set_litter AT %DB28.DBW58, 1 s
   "Box_input_counter" : Int = PLC HMI.Box_input_counter AT %DB28.DBW60, 1 s
   "Completed_pallets_counter" : Int = PLC HMI.Completed_pallets_counter AT %DB28.DBW62, 1 s
   "List_failure_and_warning" : Int = PLC HMI.List_failure_and_warning AT %DB28.DBW64, 1 s

discrete alarms
   1: 'Parada de emergencia activa en el carga paletas', class Errors, trigger "List_failure_load_pallet" bit 0
   2: 'Termico disparado en carga paletas', class Errors, trigger "List_failure_load_pallet" bit 1
   3: 'Arrancador del carga paletas fallo', class Errors, trigger "List_failure_load_pallet" bit 2
   6: 'Arrancador del alimentador de cajas fallo', class Errors, trigger "List_failure_box_feeder" bit 2
   5: 'Termico disparado en alimentador de cajas', class Errors, trigger "List_failure_box_feeder" bit 1
   4: 'Parada de emergencia activa en el alimentador de cajas', class Errors, trigger "List_failure_box_feeder" bit 0
   9: 'Arrancador del transportador de cajas fallo', class Errors, trigger "List_failure_load_beld" bit 2
   8: 'Termico disparado en el transportador de cajas', class Errors, trigger "List_failure_load_beld" bit 1
   7: 'Parada de emergencia activa en el transportador de cajas', class Errors, trigger "List_failure_load_beld" bit 0
   12: 'Arrancador del elevador fallo', class Errors, trigger "List_failure_elevator" bit 2
   11: 'Termico disparado en el elevador', class Errors, trigger "List_failure_elevator" bit 1
   10: 'Parada de emergencia activa en el elevador', class Errors, trigger "List_failure_elevator" bit 0
   15: 'Arrancador del alimentador de paletas fallo', class Errors, trigger "List_failure_pallet_feeder" bit 2
   14: 'Termico disparado en el alimentador de paletas', class Errors, trigger "List_failure_pallet_feeder" bit 1
   13: 'Parada de emergencia activa en el alimentador de paletas', class Errors, trigger "List_failure_pallet_feeder" bit 0
   18: 'Arrancador del conveyor de salida fallo', class Errors, trigger "List_failure_exit_conveyor" bit 2
   17: 'Termico disparado en conveyor de salida', class Errors, trigger "List_failure_exit_conveyor" bit 1
   16: 'Parada de emergencia activa del conveyor de salida', class Errors, trigger "List_failure_exit_conveyor" bit 0
   22: 'Valor de camada no puede ser 3', class Errors, trigger "List_failure_and_warning" bit 4
   21: 'Valor de camada no puede ser 5', class Errors, trigger "List_failure_and_warning" bit 3
   20: 'Valor de camadas debe ser menor a 7', class Errors, trigger "List_failure_and_warning" bit 2
   19: 'Valor de camadas debe ser mayor a 1', class Errors, trigger "List_failure_and_warning" bit 1

text list "Text_list_status": 0 'Palletizadora en reposo'; 1 'Manual activado'; 2 'Automatico activado'

text list "Text_list_status_motor": 0 'Motor en reposo'; 1 'Motor en movimiento'; 2 'Motor en falla'

text list "Text_list_alarms": 0 ''; 1 'Parada de emergencia activada'; 2 'Proteccion termica activada'; 3 'Problemas con la respuesta del contactor'

graphic list "Graphic_list_status": 0 'Graphic_21'; 1 'Graphic_6'; 2 'Graphic_4'

graphic list "Graphic_rotation_motor": 0 'Graphic_23'; 1 'Graphic_17'; 2 'Graphic_18'; 3 'Graphic_22'; 4 'Graphic_19'

Template "Template_1" 1280x800
   SymbolicIOField "Symbolic_IO_Field_Screen" at 25,716 size 319x53; TextOff '0'; TextOn '1'; TextList "Text_list_status"
      on Change: ActivateScreenByNumber("Tag_ScreenNumber", 0)
      ProcessValue <- "List_message"
      Appearance <- "List_message"
   TextField "Text field_1" at 484,52 size 307x62; Text 'Paletizadora'
   GraphicView "Template_Graphic view_1" at 0,0 size 196x102; Picture "floriambra._1"

screen "Main" 1280x800, template "Template_1"
   Button "Button_mode_manual" at 550,280 size 181x48; TextOff 'Modo manual'
      on Click: ActivateScreen("Manual", 0)
      on Press: function_b14e0dd5("Mode_manual", 0)
   Button "Button_mode_auto" at 550,395 size 181x49; TextOff 'Modo automatico'
      on Click: ActivateScreen("Auto", 0)
      on Press: function_b14e0dd5("Mode_Auto", 0)

screen "Auto" 1280x800, template "Template_1"
   TextField "Text field_2" at 389,141 size 533x47; Text 'Sistema en modo automatico'
   TextField "Text field_3" at 106,224 size 103x25; Text 'Punto cero'
   Button "Button_12" at 1061,706 size 181x48; TextOff 'Pantalla Principal'
      on Click: ActivateScreen("Main", 0)
      on Press: function_b14e0dd5("Mode_rest", 0)
   Rectangle "Rectangle_1" at 120,632 size 325x20
      Appearance <- "Enabled_pallet_feeder"
   Rectangle "Rectangle_2" at 445,632 size 210x20
      Appearance <- "Enabled_load_pallet"
   Rectangle "Rectangle_3" at 655,632 size 325x20
      Appearance <- "Enabled_exit_conveyor"
   Rectangle "Rectangle_5" at 121,398 size 325x20
      Appearance <- "Enabled_box_feeder"
   Rectangle "Rectangle_6" at 446,398 size 209x20
      Appearance <- "Enabled_load_beld"
   GraphicView "Graphic view_5" at 208,219 size 40x38; Picture "Graphic_5"
      Visibility <- "cero_point"
   GraphicView "Graphic view_6" at 208,219 size 40x38; Picture "Graphic_6"
      Visibility <- "cero_point"
   GraphicView "Graphic view_8" at 454,325 size 29x45; Picture "Graphic_8"
   GraphicView "Graphic view_10" at 351,326 size 52x39; Picture "Graphic_11"
   Rectangle "Rectangle_8" at 447,622 size 206x9
      VerticalMovement <- "Elevator_moving"
   TextField "Text field_4" at 429,438 size 13x18; Text '1'
   TextField "Text field_5" at 429,456 size 13x18; Text '2'
   TextField "Text field_7" at 429,477 size 13x18; Text '3'
   TextField "Text field_8" at 429,498 size 13x18; Text '4'
   TextField "Text field_9" at 429,517 size 13x18; Text '5'
   TextField "Text field_10" at 429,535 size 13x18; Text '6'
   IOField "I/O field_1" at 1110,304 size 105x32; FormatPattern 9
      ProcessValue <- "Set_litter"
   TextField "Text field_13" at 1092,270 size 139x25; Text 'Set de camadas'
   Button "Button_2" at 1062,632 size 181x48; TextOff 'Reset'
      on Press: function_b14e0dd5("Reset", 0)
   IOField "I/O field_3" at 937,303 size 105x33; FormatPattern 999
      ProcessValue <- "Box_input_counter"
   TextField "Text field_6" at 916,270 size 138x25; Text 'Cajas entrantes'
   IOField "I/O field_5" at 937,390 size 105x34; FormatPattern 999
      ProcessValue <- "Completed_pallets_counter"
   TextField "Text field_16" at 900,352 size 181x25; Text 'Paletas completadas'
   GraphicIOField "Graphic I/O field_1" at 112,421 size 49x45; PictureList "Graphic_rotation_motor"
      ProcessValue <- "Rotation_box_feeder"
   GraphicView "Graphic view_1" at 108,418 size 55x48; Picture "Graphic_4"
      Visibility <- "Failure_box_feeder"
   GraphicIOField "Graphic I/O field_2" at 97,588 size 49x45; PictureList "Graphic_rotation_motor"
      ProcessValue <- "Rotation_pallet_feeder"
   GraphicView "Graphic view_2" at 95,585 size 55x48; Picture "Graphic_4"
      Visibility <- "Failure_pallet_feeder"
   GraphicIOField "Graphic I/O field_3" at 948,584 size 49x45; PictureList "Graphic_rotation_motor"
      ProcessValue <- "Rotation_exit_conveyor"
   GraphicView "Graphic view_4" at 946,582 size 55x48; Picture "Graphic_4"
      Visibility <- "Failure_exit_conveyor"
   GraphicIOField "Graphic I/O field_4" at 389,585 size 49x45; PictureList "Graphic_rotation_motor"
      ProcessValue <- "Rotation_load_pallet"
   GraphicView "Graphic view_7" at 385,584 size 55x48; Picture "Graphic_4"
      Visibility <- "Failure_load_pallet"
   GraphicIOField "Graphic I/O field_5" at 660,567 size 49x45; PictureList "Graphic_rotation_motor"
      ProcessValue <- "Rotation_elevator"
   GraphicView "Graphic view_11" at 659,567 size 55x48; Picture "Graphic_4"
      Visibility <- "Failure_exit_conveyor"
   GraphicIOField "Graphic I/O field_6" at 644,348 size 49x45; PictureList "Graphic_rotation_motor"
      ProcessValue <- "Rotation_load_beld"
   GraphicView "Graphic view_12" at 643,346 size 55x48; Picture "Graphic_4"
      Visibility <- "Failure_load_beld"
   TextField "Text field_1" at 472,655 size 165x25; Text 'Elevador Subiendo'
      Visibility <- "Enabled_up_elevator"
      Appearance <- "Enabled_up_elevator"
   TextField "Text field_17" at 474,655 size 155x25; Text 'Elevador Bajando'
      Visibility <- "Enabled_down_elevator"
      Appearance <- "Enabled_down_elevator"
   Circle "Circle_1" at 461,336 size 16x16
      Visibility <- "Enabled_turn"
      Appearance <- "Enabled_turn"
   GraphicView "Graphic view_13" at 515,325 size 29x45; Picture "Graphic_8"
   Circle "Circle_2" at 522,336 size 16x16
      Appearance <- "Enabled_push"
      Visibility <- "Enabled_push"
   GraphicView "Graphic view_14" at 576,325 size 29x45; Picture "Graphic_8"
   Circle "Circle_3" at 583,336 size 16x16
      Appearance <- "Enabled_clamp"
      Visibility <- "Enabled_clamp"
   GraphicView "Graphic view_3" at 665,415 size 29x45; Picture "Graphic_8"
   Circle "Circle_4" at 672,426 size 16x16
      Visibility <- "Enabled_plate"
      Appearance <- "Enabled_plate"
   Circle "Circle_5" at 380,334 size 16x16
      Appearance <- "Box_counter"
      Visibility <- "Box_counter"
   TextField "Text field_11" at 449,299 size 42x20; Text 'Forma'
   TextField "Text field_12" at 506,299 size 48x20; Text 'Empuje'
   TextField "Text field_18" at 573,299 size 37x20; Text 'Regla'
   TextField "Text field_19" at 698,425 size 33x20; Text 'Plato'
   TextField "Text field_20" at 698,338 size 87x20; Text 'Transportador'
   TextField "Text field_21" at 730,353 size 19x20; Text 'de'
   TextField "Text field_22" at 722,366 size 35x20; Text 'cajas'
   TextField "Text field_23" at 29,392 size 74x20; Text 'Alimentador'
   TextField "Text field_24" at 54,406 size 19x20; Text 'de'
   TextField "Text field_25" at 45,419 size 35x20; Text 'cajas'
   TextField "Text field_26" at 21,541 size 74x20; Text 'Alimentador'
   TextField "Text field_27" at 45,554 size 19x20; Text 'de'
   TextField "Text field_28" at 31,567 size 46x20; Text 'paletas'
   TextField "Text field_29" at 327,559 size 39x20; Text 'Carga'
   TextField "Text field_30" at 336,573 size 19x20; Text 'de'
   TextField "Text field_31" at 324,586 size 46x20; Text 'paletas'
   TextField "Text field_32" at 718,540 size 54x20; Text 'Elevador'
   TextField "Text field_33" at 734,553 size 19x20; Text 'de'
   TextField "Text field_34" at 721,566 size 46x20; Text 'paletas'
   TextField "Text field_35" at 977,537 size 58x20; Text 'Conveyor'
   TextField "Text field_36" at 995,551 size 19x20; Text 'de'
   TextField "Text field_37" at 986,565 size 38x20; Text 'salida'
   TextField "Text field_38" at 358,299 size 61x20; Text 'Contador'

screen "Manual" 1280x800, template "Template_1"
   Button "Button_box_feeder_driver" at 258,272 size 181x48; TextOff 'Start'
      on Click: ActivateScreen("Drive_box_feeder", 0)
   TextField "Text field_2" at 406,142 size 463x47; Text 'Sistema en modo manual'
   TextField "Text field_3" at 252,238 size 185x25; Text 'Alimentador de cajas'
   Button "Button_load_beld_driver" at 258,377 size 181x48; TextOff 'Start'
      on Click: ActivateScreen("Drive_load_belt", 0)
   TextField "Text field_4" at 248,344 size 202x25; Text 'Transportador de cajas'
   Button "Button_elevator_driver" at 258,480 size 181x48; TextOff 'Start'
      on Click: ActivateScreen("Drive_elevator", 0)
   TextField "Text field_5" at 311,445 size 79x25; Text 'Elevador'
   Button "Button_load_pallet_driver" at 258,584 size 181x48; TextOff 'Start'
      on Click: ActivateScreen("Drive_load_pallet", 0)
   Button "Button_pallet_feeder_driver" at 570,272 size 181x48; TextOff 'Start'
      on Click: ActivateScreen("Drive_pallet_feeder", 0)
   TextField "Text field_7" at 280,549 size 138x25; Text 'Carga de paleta'
   Button "Button_exit_conveyor_driver" at 570,377 size 181x48; TextOff 'Start'
      on Click: ActivateScreen("Drive_exit_conveyor", 0)
   TextField "Text field_8" at 557,238 size 203x25; Text 'Alimentador de paletas'
   Button "Button_7" at 570,480 size 181x48; TextOff 'Start'
      on Press: function_b14e0dd5("Enable_turn", 0)
   TextField "Text field_9" at 576,344 size 167x25; Text 'Conveyor de salida'
   Button "Button_8" at 570,584 size 181x48; TextOff 'Start'
      on Press: function_b14e0dd5("Enable_push", 0)
   TextField "Text field_10" at 577,446 size 166x25; Text 'Accionador de giro'
   Button "Button_9" at 883,272 size 181x48; TextOff 'Start'
      on Press: function_b14e0dd5("Enable_clamp", 0)
   TextField "Text field_11" at 576,549 size 173x25; Text 'Empujador de cajas'
   Button "Button_10" at 883,377 size 181x48; TextOff 'Start'
      on Press: function_b14e0dd5("Enable_plate", 0)
   TextField "Text field_12" at 948,238 size 53x25; Text 'Regla'
   TextField "Text field_13" at 947,344 size 49x25; Text 'Plato'
   Button "Button_12" at 1034,697 size 181x48; TextOff 'Pantalla Principal'
      on Click: ActivateScreen("Main", 0)
      on Press: function_b14e0dd5("Mode_rest", 0)

screen "Drive_box_feeder" 1280x800, template "Template_1"
   Button "Button_1" at 427,350 size 181x48; TextOff 'Start'
      on Press: function_b14e0dd5("Start_box_feeder", 0)
   Button "Button_2" at 427,418 size 181x48; TextOff 'Stop'
      on Press: function_b14e0dd5("Stop_box_feeder", 0)
   Button "Button_3" at 427,493 size 181x48; TextOff 'Reset'
      on Press: function_b14e0dd5("Reset", 0)
   Button "Button_12" at 1034,697 size 181x48; TextOff 'Pantalla Principal'
      on Press: ActivateScreen("Manual", 0)
   GraphicView "Graphic view_5" at 344,321 size 50x42; Picture "Graphic_4"
      Visibility <- "Failure_box_feeder"
   SymbolicIOField "Symbolic I/O field_2" at 624,390 size 235x41; TextOff '0'; TextOn '1'; TextList "Text_list_status_motor"
      ProcessValue <- "Status_box_feeder"
   SymbolicIOField "Symbolic I/O field_1" at 411,294 size 470x37; TextOff '0'; TextOn '1'; TextList "Text_list_alarms"
      ProcessValue <- "List_failure_box_feeder"
   GraphicIOField "Graphic I/O field_1" at 699,439 size 87x77; PictureList "Graphic_rotation_motor"
      ProcessValue <- "Rotation_box_feeder"
   TextField "Text field_1" at 566,160 size 17x25; Text 'Text'
   TextField "Text field_2" at 442,188 size 389x47; Text 'Alimentador de cajas'

screen "Drive_load_belt" 1280x800, template "Template_1"
   Button "Button_1" at 427,350 size 181x48; TextOff 'Start'
      on Press: function_b14e0dd5("Start_load_beld", 0)
   Button "Button_2" at 427,418 size 181x48; TextOff 'Stop'
      on Press: function_b14e0dd5("Stop_load_beld", 0)
   Button "Button_3" at 427,493 size 181x48; TextOff 'Reset'
      on Press: function_b14e0dd5("Reset", 0)
   Button "Button_12" at 1034,697 size 181x48; TextOff 'Pantalla Principal'
      on Press: ActivateScreen("Manual", 0)
   GraphicView "Graphic view_5" at 344,321 size 50x42; Picture "Graphic_4"
      Visibility <- "Failure_load_beld"
   SymbolicIOField "Symbolic I/O field_2" at 624,390 size 235x41; TextOn '1'; TextOff '0'; TextList "Text_list_status_motor"
      ProcessValue <- "Status_load_beld"
   SymbolicIOField "Symbolic I/O field_1" at 411,294 size 470x37; TextOn '1'; TextOff '0'; TextList "Text_list_alarms"
      ProcessValue <- "List_failure_load_beld"
   GraphicIOField "Graphic I/O field_1" at 699,439 size 87x77; PictureList "Graphic_rotation_motor"
      ProcessValue <- "Rotation_load_beld"
   TextField "Text field_1" at 566,160 size 17x25; Text 'Text'
   TextField "Text field_2" at 442,188 size 427x47; Text 'Transportador de cajas'

screen "Drive_elevator" 1280x800, template "Template_1"
   Button "Button_1" at 427,350 size 181x48; TextOff 'Subir elevador'
      on Press: function_b14e0dd5("Up_elevator", 0)
   Button "Button_2" at 427,418 size 181x48; TextOff 'Bajar elevador'
      on Press: function_b14e0dd5("Down_elevator", 0)
   Button "Button_3" at 427,493 size 181x48; TextOff 'Reset'
      on Press: function_b14e0dd5("Reset", 0)
   Button "Button_12" at 1034,697 size 181x48; TextOff 'Pantalla Principal'
      on Press: ActivateScreen("Manual", 0)
   GraphicView "Graphic view_5" at 344,321 size 50x42; Picture "Graphic_4"
      Visibility <- "Failure_elevator"
   SymbolicIOField "Symbolic I/O field_2" at 624,390 size 235x41; TextOn '1'; TextOff '0'; TextList "Text_list_status_motor"
      ProcessValue <- "Status_elevator"
   SymbolicIOField "Symbolic I/O field_1" at 411,294 size 470x37; TextOn '1'; TextOff '0'; TextList "Text_list_alarms"
      ProcessValue <- "List_failure_elevator"
   GraphicIOField "Graphic I/O field_1" at 699,439 size 87x77; PictureList "Graphic_rotation_motor"
      ProcessValue <- "Rotation_elevator"
   TextField "Text field_1" at 566,160 size 17x25; Text 'Text'
   TextField "Text field_2" at 564,185 size 163x47; Text 'Elevador'

screen "Drive_load_pallet" 1280x800, template "Template_1"
   Button "Button_1" at 427,350 size 181x48; TextOff 'Start'
      on Press: function_b14e0dd5("Start_load_pallet", 0)
   Button "Button_2" at 427,418 size 181x48; TextOff 'Stop'
      on Press: function_b14e0dd5("Stop_load_pallet", 0)
   Button "Button_3" at 427,493 size 181x48; TextOff 'Reset'
      on Press: function_b14e0dd5("Reset", 0)
   Button "Button_12" at 1034,697 size 181x48; TextOff 'Pantalla Principal'
      on Press: ActivateScreen("Manual", 0)
   GraphicView "Graphic view_5" at 344,321 size 50x42; Picture "Graphic_4"
      Visibility <- "Failure_load_pallet"
   SymbolicIOField "Symbolic I/O field_2" at 624,390 size 235x41; TextOn '1'; TextOff '0'; TextList "Text_list_status_motor"
      ProcessValue <- "Status_load_pallet"
   SymbolicIOField "Symbolic I/O field_1" at 411,294 size 470x37; TextOn '1'; TextOff '0'; TextList "Text_list_alarms"
      ProcessValue <- "List_failure_load_pallet"
   GraphicIOField "Graphic I/O field_1" at 699,439 size 87x77; PictureList "Graphic_rotation_motor"
      ProcessValue <- "Rotation_load_pallet"
   TextField "Text field_1" at 566,160 size 17x25; Text 'Text'
   TextField "Text field_2" at 485,185 size 311x47; Text 'Carga de paletas'

screen "Drive_pallet_feeder" 1280x800, template "Template_1"
   Button "Button_1" at 427,350 size 181x48; TextOff 'Start'
      on Press: function_b14e0dd5("Start_pallet_feeder", 0)
   Button "Button_2" at 427,418 size 181x48; TextOff 'Stop'
      on Press: function_b14e0dd5("Stop_pallet_feeder", 0)
   Button "Button_3" at 427,493 size 181x48; TextOff 'Reset'
      on Press: function_b14e0dd5("Reset", 0)
   Button "Button_12" at 1034,697 size 181x48; TextOff 'Pantalla Principal'
      on Press: ActivateScreen("Manual", 0)
   GraphicView "Graphic view_5" at 344,321 size 50x42; Picture "Graphic_4"
      Visibility <- "Failure_pallet_feeder"
   SymbolicIOField "Symbolic I/O field_2" at 624,390 size 235x41; TextOn '1'; TextOff '0'; TextList "Text_list_status_motor"
      ProcessValue <- "Status_pallet_feeder"
   SymbolicIOField "Symbolic I/O field_1" at 411,294 size 470x37; TextOn '1'; TextOff '0'; TextList "Text_list_alarms"
      ProcessValue <- "List_failure_pallet_feeder"
   GraphicIOField "Graphic I/O field_1" at 699,439 size 87x77; PictureList "Graphic_rotation_motor"
      ProcessValue <- "Rotation_pallet_feeder"
   TextField "Text field_1" at 566,160 size 17x25; Text 'Text'
   TextField "Text field_2" at 436,188 size 427x47; Text 'Alimentador de paletas'

screen "Drive_exit_conveyor" 1280x800, template "Template_1"
   Button "Button_1" at 427,350 size 181x48; TextOff 'Start'
      on Press: function_b14e0dd5("Start_exit_conveyor", 0)
   Button "Button_2" at 427,418 size 181x48; TextOff 'Stop'
      on Press: function_b14e0dd5("Stop_exit_conveyor", 0)
   Button "Button_3" at 427,493 size 181x48; TextOff 'Reset'
      on Press: function_b14e0dd5("Reset", 0)
   Button "Button_12" at 1034,697 size 181x48; TextOff 'Pantalla Principal'
      on Press: ActivateScreen("Manual", 0)
   GraphicView "Graphic view_5" at 344,321 size 50x42; Picture "Graphic_4"
      Visibility <- "Failure_exit_conveyor"
   SymbolicIOField "Symbolic I/O field_2" at 624,390 size 235x41; TextOn '1'; TextOff '0'; TextList "Text_list_status_motor"
      ProcessValue <- "Status_exit_conveyor"
   SymbolicIOField "Symbolic I/O field_1" at 411,294 size 470x37; TextOn '1'; TextOff '0'; TextList "Text_list_alarms"
      ProcessValue <- "List_failure_exit_conveyor"
   GraphicIOField "Graphic I/O field_1" at 699,439 size 87x77; PictureList "Graphic_rotation_motor"
      ProcessValue <- "Rotation_exit_conveyor"
   TextField "Text field_1" at 566,160 size 17x25; Text 'Text'
   TextField "Text field_2" at 464,187 size 349x47; Text 'Conveyor de salida'
*)